(* IEC 61131-3 sources: st-mode/test, 1 file *)

(* ---- first.st ---- *)
(*
        I am an comment.
*)

TIME#2ms
BIT#1
INT#16#F

"fdsafdsafdsafsdaf "
'fdsafsafdsaf'
BIT#1
TRUE
FALSE
false
program abc

IF
a
THEN
        c := 2
END_IF

IF a THEN
        fsdaf
        IF a THEN
                c := 2
        ELSE
                a := 1
                b := 2
        END_IF
END_IF

IF aTHEN

IF a!=2 THEN
        a:=2
ELSE
        ab:=6
END_IF

END_PROGRAM
